TYPE ST_RECORD_DATA:
STRUCT
	rPosition:		    REAL;
	rPressureInBar:		REAL;
END_STRUCT
END_TYPE

(* stored: Version 1.1.0.1, ProductVersion 3.1.4024.12
   DUT ST_RECORD_DATA: Id {62a8be30-065d-431a-829f-02851b1d20c2} *)
